# EPICS IOC start-up script: iocsh/amp.iocsh
##############################################################################
####                        SSA Amplifier iocsh                            ###
##############################################################################
#- PREFIX_AMP    - Prefix used for record names
#- PREFIX_CGD    - Prefix used for CGD records
#- AMP_CHAR      - The letter of the amplifier
#- NUM_SSM       - The number of SSMs in this amplifier
#- AMP_SSM       - The list of SSMs in this amplifier, separated by commas
#-#############################################################################

dbLoadRecords("$(myrrha_ssa_DB)amp.db", "PREFIX=$(PREFIX_AMP),PREFIX_CGD=$(PREFIX_CGD),AMP_CHAR=$(AMP_CHAR),NUM_SSM=$(NUM_SSM),AMP_SSM=$(AMP_SSM)")
dbLoadRecords("$(myrrha_ssa_DB)amp_cmd.db", "PREFIX=$(PREFIX_AMP),PREFIX_CGD=$(PREFIX_CGD),AMP_CHAR=$(AMP_CHAR)")
